Universal Robots PolyScope program: presa_palla.urp

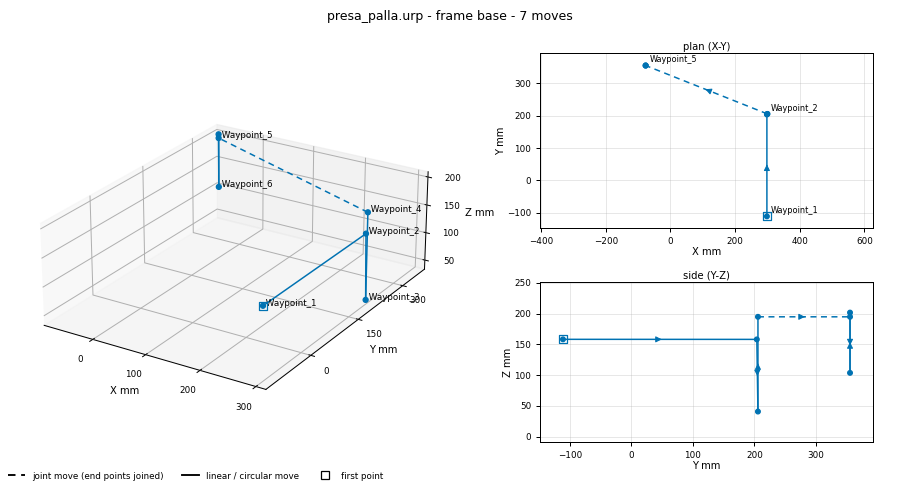
[picture p0: tool path of presa_palla.urp in frame base, 7 of 7 moves have a stored position in this frame; points joined in program order, loops and branches not executed]
Program presa_palla (installation=default directory=/programs createdIn=3.15.8.106339 lastSavedIn=3.15.8.106339 robotSerialNumber=2023330215)
Calibrated DH parameters: a=[-0.000158, -0.243568, -0.211872, 0.000029, -0.000046, 0]; d=[0.151957, 0.552568, 8.396945, -8.837237, 0.085345, 0.082393]; alpha=[1.571201, -0.003022, 0.002719, 1.570411, -1.571935, 0]; deltaTheta=[0.000034, -0.006936, 0.121129, -0.114397, -0.000018, 0.00002]
Robot Program (runOnlyOnce=false)
  MoveJ speed 60 deg/s, acceleration 80 deg/s^2 (useActiveTCP=true)
    Waypoint Waypoint_1: TCP in base x=298.404 y=-111.257 z=158.293 mm, rx=-2.784 ry=-1.4521 rz=0.0016 rad; joints [0.005, -90.001, -90.013, -90.002, 90.186, 575.047] deg; flange x=298.658 y=-111.405 z=313.292 mm, rx=-2.784 ry=-1.4521 rz=0.0016 rad
  MoveL speed 250 mm/s, acceleration 1200 mm/s^2 (useActiveTCP=true) feature=Base
    Waypoint Waypoint_2: TCP in base x=298.375 y=203.914 z=158.196 mm, rx=-2.7842 ry=-1.4522 rz=0.002 rad; joints [52.253, -100.718, -78.189, -91.047, 90.204, 627.289] deg; flange x=298.649 y=203.805 z=313.196 mm, rx=-2.7842 ry=-1.4522 rz=0.002 rad
    Waypoint Waypoint_3: TCP in base x=299.841 y=205.722 z=40.858 mm, rx=-2.7771 ry=-1.4484 rz=-0.0247 rad; joints [52.211, -107.314, -103.132, -58.43, 90.175, 627.33] deg; flange x=298.345 y=203.298 z=195.832 mm, rx=-2.7771 ry=-1.4484 rz=-0.0247 rad
    URCap SG Grip (OnRobot, OnRobot A/S)
    Waypoint Waypoint_4: TCP in base x=299.842 y=205.755 z=194.904 mm, rx=-2.777 ry=-1.4484 rz=-0.025 rad; joints [52.257, -101.085, -68.262, -99.518, 90.199, 627.27] deg; flange x=298.324 y=203.309 z=349.877 mm, rx=-2.777 ry=-1.4484 rz=-0.025 rad
  MoveJ speed 60 deg/s, acceleration 80 deg/s^2 (useActiveTCP=true)
    Waypoint Waypoint_5: TCP in base x=-76.805 y=355.454 z=194.881 mm, rx=-1.4952 ry=-2.744 rz=-0.0125 rad; joints [119.995, -101.089, -68.262, -99.518, 90.195, 627.271] deg; flange x=-75.134 y=353.126 z=349.855 mm, rx=-1.4952 ry=-2.744 rz=-0.0125 rad
  MoveL speed 250 mm/s, acceleration 1200 mm/s^2 (useActiveTCP=true) feature=Base
    Waypoint Waypoint_6: TCP in base x=-76.826 y=355.437 z=103.743 mm, rx=-1.4951 ry=-2.744 rz=-0.0125 rad; joints [119.968, -101.69, -92.209, -74.969, 90.199, 627.305] deg; flange x=-75.152 y=353.111 z=258.717 mm, rx=-1.4951 ry=-2.744 rz=-0.0125 rad
    URCap SG Release (OnRobot, OnRobot A/S) dataModel(sg-target-width-percent=100.0)
    Waypoint Waypoint_7: TCP in base x=-76.861 y=355.437 z=201.769 mm, rx=-1.4949 ry=-2.7439 rz=-0.0125 rad; joints [120.003, -101.437, -65.946, -101.478, 90.199, 627.267] deg; flange x=-75.163 y=353.102 z=356.742 mm, rx=-1.4949 ry=-2.7439 rz=-0.0125 rad
